TYPE ST_ITC_ISR :
(**************************************************************************************
 * 	Application		:	BoxControl Framework
 *	Revision		:	$Revision: 404529 $
 *	Revision date	:	$Date: 2018-04-23 08:21:38 +0200 (Mo., 23 Apr 2018) $
 *	Last changed by	:	$Author: b7bolm $
 *	URL				:	$URL: http://almscdc.swisslog.com/repo/SWPD/Development/BoxControlFramework/20_Release/trunk/01_Software/BCF/BCF/JumpStart/20_Product/10_App/11_Com/10_Lib/10_Conv/11_ITC/01_DUTs/ST_ITC_ISR.TcDUT $
 *
 *	Purpose			:	ISR Structure
 *
 * ------------------------------------------------------------------------------------
 *	Copyright Swisslog [IP AG], Switzerland. All rights reserved.
 * 
 * ------------------------------------------------------------------------------------
 *	
 * 	Revision History: 
 *
 * 	VERSION			DATE			INITIALS			DESCRIPTION
 *	0.1				01.01.2001		swl					Example
 *
 **************************************************************************************)
STRUCT
	SignalType			: INT; // 1 Digit Signal Type (0=Inputs, 1=Outputs, 2=Positions) 
	StartSignalNumber	: INT; // 4 Digit Start Signal Number 
	DataLength			: INT; // 2 Digit Data Length 
	Information			: STRING(99); // 99 Digit (HEX) Information Data 
	ReturnCode			: E_ErrorConv; // 4 Digit return code
END_STRUCT
END_TYPE

(* stored: Version 1.1.0.1, ProductVersion 3.1.4022.12
   DUT ST_ITC_ISR: Id {0eec145a-36f7-47c4-a430-e35cfcc4a9c3} *)
